(* CoDeSys 2.3.9.37 project: Cap8_6.pro *)
(* Libraries: Standard.lib 4.10.05 12:14:46 *)

(* Global variable list: Global_Variables *)
VAR_GLOBAL

      (* Entradas *)
	A: BOOL;
	B: BOOL;
      (* Salidas *)
	LuzVerde: BOOL;
	LuzAmarilla: BOOL;
	LuzRoja: BOOL;
       AvisoLleno:BOOL;

       (* Otras variables *)
       Aforo: INT;   (* Aforo máximo. Hay que darle valor *)
	Contador: CTUD;  (*Contador de  personas dentro *)
       Visitas:CTU;  (* Contados de número total de visitas *)
       Temporizador:TON; (* Temporizador para museo lleno *)

END_VAR

(* POU PLC_PRG, IL *)
PROGRAM PLC_PRG
VAR

END_VAR
	CAL		Animacion
	
END_PROGRAM

(* POU Animacion, ST *)
PROGRAM Animacion
VAR

   persona1x:INT:=-1000;
   persona1y:INT:=0;
  persona2x:INT:=-1000;
   persona2y:INT:=0;
	Ocupado: BOOL;
       EntraPersona:BOOL;
	EntrandoPersona: BOOL;
	SalePersona: BOOL;
	SaliendoPersona: BOOL;
       EntraSale:BOOL;
       EntrandoSaliendo:BOOL;
	SaleEntra: BOOL;
	SaliendoEntrando: BOOL;
       velocidad:INT:=2;
END_VAR
IF Ocupado=FALSE THEN

IF EntraPersona AND LuzRoja=FALSE THEN
   EntrandoPersona:=TRUE;
   persona1x:=0;
   Ocupado:=TRUE;
END_IF

IF SalePersona (* AND Contador.CV>0*)  THEN
   SaliendoPersona:=TRUE;
   persona2x:=0;
   Ocupado:=TRUE;
END_IF

IF EntraSale AND LuzRoja=FALSE (*AND Contador.CV>0*) THEN
   EntrandoSaliendo:=TRUE;
   persona1x:=30;
   persona2x:=0;
   Ocupado:=TRUE;
END_IF

IF SaleEntra AND LuzRoja=FALSE (*AND Contador.CV>0*) THEN
   SaliendoEntrando:=TRUE;
   persona1x:=0;
   persona2x:=-10;
   Ocupado:=TRUE;
END_IF

END_IF



IF EntrandoPersona THEN
    persona1x:=persona1x+velocidad;
    IF persona1x>70 AND persona1x<97 THEN
      A:=TRUE;
    ELSE
       A:=FALSE;
    END_IF
    IF persona1x>=75 AND persona1x<105 THEN
      B:=TRUE;
    ELSE
       B:=FALSE;
    END_IF
   IF persona1x>150 THEN
      EntrandoPersona:=FALSE;
      persona1x:=-1000;
      Ocupado:=FALSE;
   END_IF
 END_IF


IF SaliendoPersona THEN
    persona2x:=persona2x-velocidad;
    IF persona2x<-60 AND persona2x>-87 THEN
      B:=TRUE;
    ELSE
       B:=FALSE;
    END_IF
    IF persona2x<=-65 AND persona2x>-95 THEN
      A:=TRUE;
    ELSE
       A:=FALSE;
    END_IF
   IF persona2x<-150 THEN
      SaliendoPersona:=FALSE;
      persona2x:=-1000;
      Ocupado:=FALSE;
   END_IF
 END_IF


IF EntrandoSaliendo OR SaliendoEntrando THEN

    persona2x:=persona2x-velocidad;
    persona1x:=persona1x+velocidad;
    IF (persona2x<-60 AND persona2x>-87) OR (  persona1x>=75 AND persona1x<105) THEN
      B:=TRUE;
    ELSE
       B:=FALSE;
    END_IF
    IF(persona2x<=-65 AND persona2x>-95) OR ( persona1x>70 AND persona1x<97) THEN
      A:=TRUE;
    ELSE
       A:=FALSE;
    END_IF

   IF (persona2x<-150) AND (persona1x>150)  THEN
      EntrandoSaliendo:=FALSE;
     SaliendoEntrando:=FALSE;
       persona1x:=-1000;
      persona2x:=-1000;
      Ocupado:=FALSE;
   END_IF
 END_IF
END_PROGRAM

(* Visualisation Museo
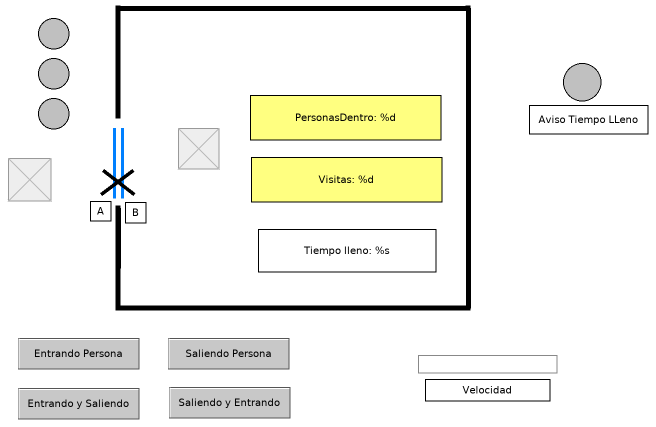
ellipse at (50,40)-(81,71): alarm colour if LuzRoja
ellipse at (50,80)-(81,111): alarm colour if LuzAmarilla
ellipse at (50,120)-(81,151): alarm colour if LuzVerde
rectangle at (262,117)-(453,162): text "PersonasDentro: %d"; shows contador.CV
bitmap at (20,180)-(61,221): SILHOUETTE_MAN_WALKING_BACKPACK.TIF
polyline at (126,150)-(126,220): alarm colour if A
polyline at (134,150)-(134,220): alarm colour if B
rectangle at (102,223)-(123,243): text "A"
rectangle at (137,224)-(158,245): text "B"
button at (30,360)-(151,391): text "Entrando Persona"; taps Animacion.EntraPersona
bitmap at (190,150)-(231,191): DibujosEj6\persona2.bmp
button at (180,360)-(301,391): text "Saliendo Persona"; taps Animacion.SalePersona
button at (30,410)-(151,441): text "Entrando y Saliendo"; taps Animacion.EntraSale
button at (181,409)-(302,440): text "Saliendo y Entrando"; taps Animacion.SaleEntra
rectangle at (437,401)-(562,423): text "Velocidad"
polyline at (115,192)-(146,216): alarm colour if LuzRoja
polyline at (113,192)-(145,216): alarm colour if luzroja
rectangle at (263,179)-(454,224): text "Visitas: %d"; shows visitas.CV
bitmap at (20,180)-(63,223): DibujosEj6\persona1.bmp
ellipse at (575,85)-(613,123): alarm colour if AvisoLleno
rectangle at (541,127)-(660,156): text "Aviso Tiempo LLeno"
rectangle at (270,251)-(448,294): text "Tiempo lleno: %s"; shows Temporizador.ET
2 more shapes without text or variables
*)
